FUNCTION_BLOCK FB_CalCulateAccumulation
VAR_INPUT
	lrAccumulator : LREAL  := 0;
	
END_VAR
VAR_OUTPUT
	accumulatedValueOut : LREAL;// value = lrAccumulator(timeNew) - lrAccumulator(timeOld)
	previousTimestampOut	: TIMESTRUCT;// TimeOld
	bNewPeriodAlarm : BOOL;// Remain True in 30s if not be ackNowledge
	
END_VAR
VAR

	
	eCpHour		: E_CompareTime;
	eCpDay 		: E_CompareTime;
	eCpMonth	: E_CompareTime;
	eCpYear		: E_CompareTime;
	eCpMinute	: E_CompareTime;
	eSameTime : E_CompareTime;
	eNewTime : E_CompareTime;
	eRfTimeCompare : REFERENCE TO E_CompareTime;
	sName 		: STRING;
	eState : UINT;
	TonRemainOutput : TON;
	eTimeAccumulate : E_CompareTime;
	bInit : BOOL;
	bReset : BOOL;
END_VAR

VAR PERSISTENT 
	bUpdatedValueLastHour : BOOL;
	previousTimestamp	: TIMESTRUCT;
	ValueInLastTime : LREAL;
	accumulatedValue : LREAL;
	
	
END_VAR
VAR CONSTANT
	eStateUinitialized : UINT := 0;
	eStateInit : UINT := 10;
	eStateRun : UINT := 20;
	eStateReset : UINT := 100;
	TimeNewPeriodAlarm : TIME := T#30s;
END_VAR



				
CASE eState OF
	eStateUinitialized: // unInitialized
		;// will go to eStateInit if MR_Run is called 
		
	eStateInit: 
		;// will call by MR_Init
		
	eStateRun: //StateRun
		MS_Run();
		
	eStateReset :
		MS_Reset();
	
END_CASE

IF eState > 0 AND bReset THEN
	eState := eStateReset;
END_IF

PROPERTY isInitDone : bool
GET
END_GET
END_PROPERTY

PROPERTY isRuning : bool
GET
isRuning := eState = eStateRun;
END_GET
END_PROPERTY

// if not return true , check the Current time and PreviousTime in fb
METHOD MR_Acknowledge : BOOL
VAR_INPUT
END_VAR
bNewPeriodAlarm := FALSE;
IF eRfTimeCompare = eSameTime THEN
	MR_Acknowledge := TRUE;
END_IF
END_METHOD

METHOD MR_Init : BOOL
VAR_INPUT
END_VAR

IF eState = eStateUinitialized THEN// init;
	bInit := true;
 
	IF MS_Init() THEN
		MR_Init := TRUE;
		eState := eStateRun;
	END_IF


END_IF
END_METHOD

METHOD MR_Reset : BOOL
VAR_INPUT
END_VAR
bReset := TRUE;
IF eState = eStateUinitialized THEN
	MR_Reset := TRUE;
	bReset := false;
END_IF
END_METHOD

METHOD Protected MS_Init : BOOL
VAR_INPUT
END_VAR
CASE eTimeAccumulate OF
	NEW_MINUTE :
		eSameTime := SAME_MINUTE;
		eNewTime := NEW_MINUTE;
		eRfTimeCompare REF= eCpMinute;
		MS_Init := TRUE;
	NEW_HOUR :
		eSameTime := SAME_HOUR;
		eNewTime := NEW_HOUR;
		eRfTimeCompare REF= eCpHour;
		MS_Init := TRUE;
	NEW_DAY	:
		eSameTime := SAME_DAY;
		eNewTime := NEW_DAY;
		eRfTimeCompare REF= eCpDay;
		MS_Init := TRUE;
	NEW_MONTH:
		eSameTime := SAME_MONTH;
		eNewTime := NEW_MONTH;
		eRfTimeCompare REF= eCpMonth;
		MS_Init := TRUE;
	NEW_YEAR:
		eSameTime := SAME_YEAR;
		eNewTime := NEW_YEAR;
		eRfTimeCompare REF= eCpYear;
		MS_Init := true;
END_CASE
END_METHOD

METHOD protected MS_Reset : BOOL
VAR_INPUT
END_VAR
//retainvalue
	
	bUpdatedValueLastHour := FALSE;
	previousTimestamp.wYear := 0;
	previousTimestamp.wMonth := 0;
	previousTimestamp.wDay := 0;
	previousTimestamp.wMinute := 0;
	previousTimestamp.wSecond := 0;
	previousTimestamp.wMilliseconds := 0;
	ValueInLastTime := 0 ;
	accumulatedValue := 0 ;
// out_put
	accumulatedValueOut := 0;
	previousTimestampOut.wYear := 0;
	previousTimestampOut.wMonth := 0;
	previousTimestampOut.wDay := 0;
	previousTimestampOut.wMinute := 0;
	previousTimestampOut.wSecond := 0;
	previousTimestampOut.wMilliseconds := 0;
	bNewPeriodAlarm := false;// Remain True 
	
// 	RETURN TO uninit
	eState := eStateUinitialized;
	eRfTimeCompare REF= 0;
END_METHOD

METHOD Protected MS_Run : BOOL
VAR_INPUT
END_VAR
	CompareTime(	timestruct1 := previousTimestamp,
					timestruct2 := GVL.fbMachineTime.systemTime,
					eCpMinute => eCpMinute, 
					eCpHour => eCpHour,
					eCpDay => eCpDay,
					eCpMonth => eCpMonth,
					ecpYear => eCpYear);

	IF eRfTimeCompare = eNewTime THEN
		// update to output
		accumulatedValueOut := accumulatedValue;
		previousTimestampOut := previousTimestamp;
		bNewPeriodAlarm := TRUE;
		// update the the last hour and time
		bUpdatedValueLastHour := FALSE;
		ValueInLastTime := lrAccumulator;
		previousTimestamp := GVL.fbMachineTime.systemTime;
		// UpdateOK
		bUpdatedValueLastHour := TRUE;
	
	ELSIF eRfTimeCompare = eSameTime AND bUpdatedValueLastHour THEN

		accumulatedValue := lrAccumulator - ValueInLastTime;
		
	ELSIF eRfTimeCompare = eSameTime AND NOT bUpdatedValueLastHour THEN
		ValueInLastTime := lrAccumulator;
		previousTimestamp := GVL.fbMachineTime.systemTime;
	ELSE
		; //invalid time Compare
	

	END_IF
	
TonRemainOutput( IN := bNewPeriodAlarm , PT := TimeNewPeriodAlarm);

IF TonRemainOutput.Q THEN
	bNewPeriodAlarm := false;
END_IF
END_METHOD

PROPERTY Name : string
GET
Name := sName;
END_GET
SET
sName := Name;
END_SET
END_PROPERTY

// Set TimeAccumulate before call Mr_Init.
//NEW_MINUTE := 5,
//	NEW_HOUR := 10,
//	NEW_DAY	:= 20,
//	NEW_MONTH := 30,
//	NEW_YEAR	:= 32,
PROPERTY TimeAccumulate : E_CompareTime
GET
TimeAccumulate := eTimeAccumulate;
END_GET
SET
eTimeAccumulate := TimeAccumulate;
END_SET
END_PROPERTY

END_FUNCTION_BLOCK

(* stored: Version 1.1.0.1, ProductVersion 3.1.4024.12
   POU FB_CalCulateAccumulation: Id {e88953d9-7557-4b87-8986-671bc8cacda9}, SpecialFunc None
   Property isInitDone: Id {baf29f36-37e5-4e03-90a8-83acb758cae9}
   Get Get: Id {eb1ad9fa-b80f-496a-9e0c-294f7bb30f95}
   Property isRuning: Id {b0bffff6-c7a7-487b-9954-eb6741969d1a}
   Get Get: Id {b9b38cce-1f09-4b53-94d5-da13439867d4}
   Method MR_Acknowledge: Id {758632cb-c0d1-4204-89c0-e713343b43f8}
   Method MR_Init: Id {9e0ff53d-25f9-442f-9ae5-85a3c64ef9dc}
   Method MR_Reset: Id {db93c866-278c-46e2-90da-71947c36fb51}
   Method MS_Init: Id {5248e55c-70a7-4639-8b20-338840b96134}
   Method MS_Reset: Id {1ebd03bb-62e3-4baf-815b-eb3a5bff8e1f}
   Method MS_Run: Id {425779c7-a7a9-4d89-ac4b-70b3443dfd76}
   Property Name: Id {da2c83d9-017c-4216-91ff-fe91f8ac4eea}
   Get Get: Id {6250de71-2f33-43bc-9325-7a078cb8ea5a}
   Set Set: Id {9531a019-6e38-4ef9-a2fa-bfd5c6d8d7bd}
   Property TimeAccumulate: Id {d51af6cd-efa0-4798-aa7e-b0c560f53e33}
   Get Get: Id {fc144cbe-4c90-465f-9bb0-f544acf6053d}
   Set Set: Id {e26844f1-07ec-44bd-abf0-a3fecb54d0a1} *)
